FUNCTION F_TO_STRING : STRING
VAR_INPUT
	Value			: ANY;
END_VAR

VAR
	pWord     : POINTER TO WORD;
END_VAR

IF Value.TypeClass = __SYSTEM.TYPE_CLASS.TYPE_WORD THEN 

	pWord := Value.pValue;
	
	F_TO_STRING := TO_STRING(pWord^);
	
	IF pWord^ < 10 THEN
		CONCAT('0',F_TO_STRING);	
	END_IF

END_IF

END_FUNCTION

(* stored: Version 1.1.0.1
   POU F_TO_STRING: Id {1568ac67-5c83-4745-9672-cd956862a2e8}, SpecialFunc None *)
